FUNCTION_BLOCK AnalogDevice IMPLEMENTS I_AnalogDevice
VAR
	Q AT%Q* : INT;
	rampUp		: RampUp;
	rampDown	: RampDown;
	_value		: REAL;
	_zeroIn		: REAL;
	_zeroOut    : REAL;
	_spanIn     : REAL;
	_spanOut    : REAL;
	_PLC_CYCLE_TIME_ms	: REAL;
	
END_VAR


	Q	:=	REAL_TO_INT(_value);

METHOD DecreaseValue
VAR_INPUT
	EN			: BOOL;
	RampDownTime: TIME;
END_VAR

	rampDown(
		IN					:= EN, 
		RampDownTime		:= RampDownTime, 
		Ramp_lowerLimit		:= _spanIn, 
		Ramp_upperLimit		:= _spanOut, 
		PLC_CYCLE_TIME_ms	:= _PLC_CYCLE_TIME_ms,
		output				:= _value, 
		InProgress			=> );
END_METHOD

METHOD FB_init : BOOL
VAR_INPUT
	bInitRetains : BOOL; // if TRUE, the retain variables are initialized (warm start / cold start)
	bInCopyCode : BOOL;  // if TRUE, the instance afterwards gets moved into the copy code (online change)
	ZeroIn		: REAL;
	ZeroOut    : REAL;
	SpanIn     : REAL;
	SpanOut    : REAL;	
	PLC_CYCLE_TIME_ms: REAL;
END_VAR

	_zeroIn		:=	ZeroIn;
	_zeroOut    :=	ZeroOut;
	_spanIn     :=	SpanIn;
	_spanOut    :=	SpanOut;
	_PLC_CYCLE_TIME_ms	:=	PLC_CYCLE_TIME_ms;
END_METHOD

METHOD IncreaseValue
VAR_INPUT
	EN			: BOOL;
	RampUpTime	: TIME;
END_VAR

	rampUp(
		IN					:= EN, 
		RampUpTime			:= RampUpTime, 
		Ramp_lowerLimit		:= _spanIn, 
		Ramp_upperLimit		:= _spanOut, 
		PLC_CYCLE_TIME_ms	:= _PLC_CYCLE_TIME_ms,
		output				:= _value, 
		InProgress			=> );
END_METHOD

METHOD Off
VAR_INPUT
END_VAR

	_value	:=	_spanIn;
END_METHOD

METHOD On
VAR_INPUT
END_VAR

	_value	:=	_spanOut;
END_METHOD

METHOD SetValue
VAR_INPUT
	value: INT;

END_VAR

	_value	:=	F_Scaling(Variable_In:= value, ZeroIn:= _zeroIn, ZeroOut:= _zeroOut, SpanIn:= _spanIn, SpanOut:= _spanOut);
END_METHOD

PROPERTY Status : INT
GET

	Status	:=	REAL_TO_INT(F_Scaling(Variable_In:= _value, ZeroIn:= _spanIn, ZeroOut:= _spanOut, SpanIn:= _zeroIn, SpanOut:= _zeroOut));
END_GET
END_PROPERTY

END_FUNCTION_BLOCK

(* stored: Version 1.1.0.1, ProductVersion 3.1.4024.13
   POU AnalogDevice: Id {c442d9c8-5ee8-45ea-97d0-22124fe9e706}, SpecialFunc None
   Method DecreaseValue: Id {4eba8c94-9dee-44a6-b5e8-6c8b6064f301}
   Method FB_init: Id {003a752a-4da4-4287-915a-505988ac7ecd}
   Method IncreaseValue: Id {15112a7c-fc96-40df-bbb2-8e365244a14c}
   Method Off: Id {68953da3-564c-4239-86ef-d3e3f467eb62}
   Method On: Id {d5657f3d-1fd6-452f-8236-c5c5b23cfe75}
   Method SetValue: Id {77141b45-bcea-4283-a002-3c6c1008b971}
   Property Status: Id {9cc97bdd-d5b5-4fa6-9e4b-03986a7d7beb}
   Get Get: Id {8e2f5ec1-13d9-4de3-8af7-1c1ea09ebd69} *)
